{attribute 'enable_dynamic_creation'}
FUNCTION_BLOCK FB_PieceSlot EXTENDS FB_Slot
VAR_INPUT
END_VAR
VAR_OUTPUT
END_VAR
VAR
	rDepth	 : REAL;
END_VAR

PROPERTY P_rDepth : REAL
GET
P_rDepth := rDepth;
END_GET
SET
rDepth := P_rDepth;
END_SET
END_PROPERTY

PROPERTY P_pPiece : POINTER TO FB_PieceBase
GET
IF pChild > 0 THEN
	P_pPiece := pChild;
END_IF
END_GET
SET
IF P_pPiece > 0 THEN
	pChild := P_pPiece;
ELSE
	pChild := 0;	
END_IF
END_SET
END_PROPERTY

END_FUNCTION_BLOCK

(* stored: Version 1.1.0.1, ProductVersion 3.1.4020.12
   POU FB_PieceSlot: Id {d9e797f4-361d-4ee7-b25d-864d9e5b00f9}, SpecialFunc None
   Property P_rDepth: Id {8078a9d9-6f8a-47a4-ad86-ccdc7bdc97fd}
   Get Get: Id {366aabd4-f8a1-43bb-bba8-08d764eaf43c}
   Set Set: Id {b5868f01-e60b-4985-a732-5453c67a9aea}
   Property P_pPiece: Id {c6532fc7-46a6-4cb9-8df0-8b5df4893901}
   Get Get: Id {be5de486-b3f3-4e00-9b71-b86d12982d26}
   Set Set: Id {c07aa166-69b8-49c2-8b44-691f93616303} *)
